TYPE ST_ShutterControl :
STRUCT

    {attribute 'pytmc' := '
        pv: REQ
        io: io
        field: DESC LSS Shutter Open Request
    '}
    bOpenRequest AT %Q* : BOOL;
    {attribute 'pytmc' := '
        pv: OPN
        io: i
        field: DESC LSS Shutter Open
    '}
    bOpenStatus AT %I* : BOOL;
    {attribute 'pytmc' := '
        pv: CLS
        io: i
        field: DESC LSS Shutter Closed
    '}
    bCloseStatus AT %I* : BOOL;
    {attribute 'pytmc' := '
        pv: LSS
        io: i
        field: DESC LSS Permission Status
    '}
    bLssStatus AT %I* : BOOL;

END_STRUCT
END_TYPE

(* stored: Version 1.1.0.1, ProductVersion 3.1.4022.18
   DUT ST_ShutterControl: Id {b813667e-4e01-43d7-9664-bdcec5c66635} *)
